(*
This file is present, but not yet tracked in the PLC project file.
*)
FUNCTION_BLOCK FB_Untracked
VAR_INPUT
END_VAR
VAR_OUTPUT
END_VAR
VAR
END_VAR

END_FUNCTION_BLOCK

(* stored: Version 1.1.0.1, ProductVersion 3.1.4024.11
   POU FB_Untracked: Id {efb8ac47-2fe7-4283-8729-6975cbd93c8f}, SpecialFunc None *)
